{attribute 'GeneratedUsingTerminal: EL5122-0000-0016'}
{attribute addProperty BoxType "EL5122-0000-0016"}
{attribute addProperty Id "EtcSlaveTerminalBaseENC_Status_Channel_1AT %I*ENC_Status_Channel_04F16FC020ENC_Status_Channel_2AT %I*ENC_Status_Channel_04F16FC020ENC_Control_Channel_1AT %Q*ENC_Control_Channel_B930862D10ENC_Control_Channel_2AT %Q*ENC_Control_Channel_B930862D10WcStateAT %I*WcState_9091E0EB2InfoDataAT %I*InfoData_32EB74EA10"}
{attribute addProperty CRC "652093243"}
{attribute addProperty Size "72"}
TYPE EL5122_26DE273B EXTENDS EtcSlaveTerminalBase :
STRUCT
	{attribute addProperty Name "ENC_Status_Channel_1"}
	ENC_Status_Channel_1 : ENC_Status_Channel_04F16FC0;
	{attribute addProperty Name "ENC_Status_Channel_2"}
	ENC_Status_Channel_2 : ENC_Status_Channel_04F16FC0;
	{attribute addProperty Name "ENC_Control_Channel_1"}
	ENC_Control_Channel_1 : ENC_Control_Channel_B930862D;
	{attribute addProperty Name "ENC_Control_Channel_2"}
	ENC_Control_Channel_2 : ENC_Control_Channel_B930862D;
	{attribute addProperty Name "WcState"}
	WcState : WcState_9091E0EB;
	{attribute addProperty Name "InfoData"}
	InfoData : InfoData_32EB74EA;
END_STRUCT
END_TYPE

(* stored: Version 1.2.0.0, ProductVersion 3.1.4024.9
   DUT EL5122_26DE273B: Id {5c1ad583-9dea-4e82-933e-ab4e35a09b36} *)
